PROGRAM Stn052_26_Stn121MainMergePrestop
VAR
	//correct
	{attribute 'TcLinkToOSO' := '.iPuckPresent   :=  <0,1,2>TIIB[N26S00 (AL1332)]^N26S02 (AL2341)^TxPDO^input byte 0;
								 .iBufferFull  :=  <0,1,2>TIIB[N26S00 (AL1332)]^N26S02 (AL2341)^TxPDO^input byte 2;
								 .oStopLower   :=  <0,1,1>TIIB[N26S00 (AL1332)]^N26S05 (EX260)^RxPDO^output byte 2'}	
	fbConvStop: FB_ConvStop;
END_VAR

//  This code instantiates a component that is implimented as a common function block
//    Note that I/O is linked directly to I/O variables inside the named instance

gStn052_26_Stn121MainMergePrestop.ConvRunning  := gConsumed_SafetyInterfaceConv.MtrRunning.Enc054Mtr07;

fbConvStop(
	pStn := ADR(gStn052),
	pCmp := ADR(gStn052_26_Stn121MainMergePrestop),
	pUpstreamStop := 0,
	pStateTraceBuffer := ADR(gStn052_StateTraceBuffer),
	pStateTraceFifo := ADR(gStn052_StateTraceFifo),
	pStats := ADR(gStn052_02_Stats));

END_PROGRAM

(* stored: Version 1.1.0.1, ProductVersion 3.1.4024.6
   POU Stn052_26_Stn121MainMergePrestop: Id {42dc5bc5-0724-449d-8b14-8f4e408a7675}, SpecialFunc None *)
